// Sets the boolean value to false if it is true and returns true if it was true before being set.
FUNCTION F_ResetOnTrue  : BOOL // Whether the value was true before resetting.
VAR_INPUT
	bValue : REFERENCE TO BOOL; // Boolean value to reset.
END_VAR

F_ResetOnTrue 	:= bValue;
bValue 			:= FALSE;

END_FUNCTION

(* stored: Version 1.1.0.1, ProductVersion 3.1.4024.15
   POU F_ResetOnTrue: Id {729735ce-5665-4b8d-ba92-5661cda9c9d4}, SpecialFunc None *)
